(* PLC project line_large.project, CODESYS CODESYS V3.5 SP22 Patch 3 *)
(* stored: creationDateTime 2026-09-17T16:10:53.5685257, modificationDateTime 2026-09-17T16:10:22.7280689 *)

PROGRAM PLC_PRG
  VAR
    fbConv1 : FB_Motor;  (* Băng tải 1 *)
    fbConv2 : FB_Motor;  (* Băng tải 2 *)
    fbConv3 : FB_Motor;  (* Băng tải 3 *)
    bLineReady : BOOL;  (* Dây chuyền sẵn sàng *)
  END_VAR

                    bLineReady := bEStopOK AND bDoorClosed AND bAutoMode;

fbConv1(bStart := bStart1, bStop := bStop1, bFault := bFault1, bInterlock := bLineReady, bRun => bMotor1);
fbConv2(bStart := bStart2, bStop := bStop2, bFault := bFault2, bInterlock := bLineReady AND bMotor1, bRun => bMotor2);
fbConv3(bStart := bStart3, bStop := bStop3, bFault := bFault3, bInterlock := bLineReady AND bMotor2, bRun => bMotor3);

rTankLevel := FC_Scale(iRaw := iTankLevelRaw, rMin := 0.0, rMax := 100.0);
rTemp      := FC_Scale(iRaw := iTempRaw, rMin := -20.0, rMax := 150.0);

bLampAlarm := fbConv1.bAlarm OR fbConv2.bAlarm OR fbConv3.bAlarm OR NOT bEStopOK;
iSpeedRef  := REAL_TO_INT(rTankLevel * 276.48);

PRG_Alarm();
                  
END_PROGRAM

FUNCTION_BLOCK FB_Motor
  VAR_INPUT
    bStart : BOOL;  (* Lệnh chạy *)
    bStop : BOOL;  (* Lệnh dừng (NC) *)
    bFault : BOOL;  (* Tín hiệu lỗi *)
    bInterlock : BOOL;  (* Điều kiện cho phép chạy *)
  END_VAR
  VAR_OUTPUT
    bRun : BOOL;  (* Lệnh ra contactor *)
    bAlarm : BOOL;  (* Báo lỗi *)
  END_VAR
  VAR
    tonFault : TON;  (* Lọc nhiễu tín hiệu lỗi *)
  END_VAR

                    tonFault(IN := bFault, PT := T#500MS);
bAlarm := tonFault.Q;
bRun := (bStart OR bRun) AND bStop AND bInterlock AND NOT bAlarm;
                  
END_FUNCTION_BLOCK

FUNCTION FC_Scale : REAL
  VAR_INPUT
    iRaw : INT;  (* Giá trị analog thô *)
    rMin : REAL;  (* Giá trị kỹ thuật nhỏ nhất *)
    rMax : REAL;  (* Giá trị kỹ thuật lớn nhất *)
  END_VAR

                    FC_Scale := rMin + (INT_TO_REAL(iRaw) / 27648.0) * (rMax - rMin);
                  
END_FUNCTION

PROGRAM PRG_Alarm

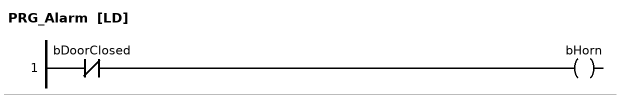
(* LD diagram, written out as Structured Text *)

bHorn := NOT bDoorClosed;
END_PROGRAM

CONFIGURATION Device
  RESOURCE Application ON PLC
    VAR_GLOBAL  (* GVL_IO *)
      bStart1 AT %IX0.0 : BOOL;  (* Start băng tải 1 *)
      bStop1 AT %IX0.1 : BOOL;  (* Stop băng tải 1 (NC) *)
      bFault1 AT %IX0.2 : BOOL;  (* Quá tải băng tải 1 *)
      bStart2 AT %IX0.3 : BOOL;  (* Start băng tải 2 *)
      bStop2 AT %IX0.4 : BOOL;  (* Stop băng tải 2 (NC) *)
      bFault2 AT %IX0.5 : BOOL;  (* Quá tải băng tải 2 *)
      bStart3 AT %IX0.6 : BOOL;  (* Start băng tải 3 *)
      bStop3 AT %IX0.7 : BOOL;  (* Stop băng tải 3 (NC) *)
      bFault3 AT %IX1.0 : BOOL;  (* Quá tải băng tải 3 *)
      bEStopOK AT %IX1.1 : BOOL;  (* Mạch dừng khẩn bình thường *)
      bDoorClosed AT %IX1.2 : BOOL;  (* Cửa tủ đã đóng *)
      iTankLevelRaw AT %IW10 : INT;  (* Mức bồn, analog thô *)
      iTempRaw AT %IW12 : INT;  (* Nhiệt độ, analog thô *)
      bMotor1 AT %QX0.0 : BOOL;  (* Contactor băng tải 1 *)
      bMotor2 AT %QX0.1 : BOOL;  (* Contactor băng tải 2 *)
      bMotor3 AT %QX0.2 : BOOL;  (* Contactor băng tải 3 *)
      bLampAlarm AT %QX0.3 : BOOL;  (* Đèn báo lỗi *)
      bHorn AT %QX0.4 : BOOL;  (* Còi báo *)
      iSpeedRef AT %QW10 : INT;  (* Tốc độ đặt cho biến tần *)
      bAutoMode AT %MX0.0 : BOOL;  (* Chế độ tự động *)
      rTankLevel : REAL;  (* Mức bồn (%) *)
      rTemp : REAL;  (* Nhiệt độ (°C) *)
    END_VAR
    TASK MainTask(INTERVAL := T#20ms, PRIORITY := 1);
    PROGRAM PLC_PRG WITH MainTask : PLC_PRG;
  END_RESOURCE
END_CONFIGURATION
